FUNCTION_BLOCK ALI_D_FF_HYS (* Data latch (d) flip flop with a Hysteresis *)
  (* Standard: 61499-1 Annex A; Description: Copyright (c) 2017 fortiss GmbH, HR Agrartechnik GmbH This program and the accompanying materials are made available under the terms of the Eclipse Public License 2.0 which is available at https://www.eclipse.org/legal/epl-2.0/ SPDX-License-Identifier: EPL-2.0 *)
  (* Version 1.0, 2026-05-15, Franz Höpfinger, HR Agrartechnik GmbH, Initial Version *)
  PACKAGE adapter::events::unidirectional;
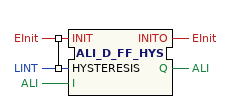
  EVENT_INPUT
    INIT : EInit WITH HYSTERESIS; (* Set Hysteresis *)
  END_EVENT
  EVENT_OUTPUT
    INITO : EInit; (* Init Confirmation *)
  END_EVENT
  VAR_INPUT
    HYSTERESIS : LINT; (* Hysteresis band *)
  END_VAR
  SOCKETS
    I : adapter::types::unidirectional::ALI; (* Value to latch *)
  END_SOCKETS
  PLUGS
    Q : adapter::types::unidirectional::ALI; (* Latched value *)
  END_PLUGS
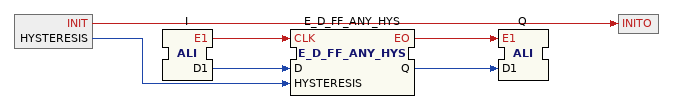
  FBS
    E_D_FF_ANY_HYS : logiBUS::signalprocessing::hysteresis::E_D_FF_ANY_HYS;
  END_FBS
  EVENT_CONNECTIONS
    I.E1 TO E_D_FF_ANY_HYS.CLK;
    E_D_FF_ANY_HYS.EO TO Q.E1;
    INIT TO INITO;
  END_CONNECTIONS
  DATA_CONNECTIONS
    I.D1 TO E_D_FF_ANY_HYS.D;
    E_D_FF_ANY_HYS.Q TO Q.D1;
    HYSTERESIS TO E_D_FF_ANY_HYS.HYSTERESIS;
  END_CONNECTIONS
END_FUNCTION_BLOCK
